(* CoDeSys 2.3.9.41 project: complex.pro *)
(* Libraries: ComService.lib 12.2.21 13:39:42, SysLibCom.lib 12.2.21 13:35:47, ModBus.lib 12.2.21 13:36:21, Util.lib 18.5.10 15:14:28, STANDARD.LIB 4.10.05 11:14:46, IECSFC.LIB 13.4.06 15:51:28, SYSLIBTIME.LIB 12.2.21 13:34:31, SYSTASKINFO.LIB 20.2.06 13:31:38, ANALYZATION.LIB 5.10.99 09:05:06, SYSLIBCALLBACK.LIB 20.2.06 13:31:08 *)

(* PLC configuration (modules and I/O channels)
Discrete input 8 bit [ID100] node 0, in %IB0 out %QB0 {Filtrationtime = 10; Filtrationtime = 10; Filtrationtime = 10; Filtrationtime = 10; Filtrationtime = 10; Filtrationtime = 10; Filtrationtime = 10; Filtrationtime = 10; Visibility = No; PinCount = 8; WatchDogPeriod = 1000; PollPeriod = 1}
  AT %IB0.0 [ByteInput] 8 discrete inputs
Discrete output - relay [ID102] node 1, in %IB1 out %QB1 {PinCount = 1; SafeValueBool = FALSE; Visibility = No}
  AT %QX1.0 [BitOutput] relay
Discrete output - relay [ID102] node 2, in %IB2 out %QB2 {PinCount = 1; SafeValueBool = FALSE; Visibility = No}
  AT %QX2.0 [BitOutput] relay
Discrete output - relay [ID102] node 3, in %IB3 out %QB3 {PinCount = 1; SafeValueBool = FALSE; Visibility = No}
  AT %QX3.0 [BitOutput] relay
Discrete output - relay [ID102] node 4, in %IB4 out %QB4 {PinCount = 1; SafeValueBool = FALSE; Visibility = No}
  AT %QX4.0 [BitOutput] relay
Discrete output - relay [ID102] node 5, in %IB5 out %QB5 {PinCount = 1; SafeValueBool = FALSE; Visibility = No}
  AT %QX5.0 [BitOutput] relay
Discrete output - relay [ID102] node 6, in %IB6 out %QB6 {PinCount = 1; SafeValueBool = FALSE; Visibility = No}
  AT %QX6.0 [BitOutput] relay
AT %QX7.0 [BitOutput] Special output
*)

(* Global variable list: Global_Variables *)
VAR_GLOBAL
	port_opened:  BYTE := 0;
	Settings:COMSETTINGS;
      	com_num: PORTS:=0;
	COM_SERVICE1: COM_SERVICE;

	port_opened2:  BYTE := 0;
	Settings2:COMSETTINGS;
      	com_num2: PORTS:=1;
	COM_SERVICE2: COM_SERVICE;


	ModBusWriteMultiReg232: MB_WR_REGS;
      ModBusReadHoldReg232: ARRAY[0..10] OF MB_RD_HOLD_REGS;
	TonConnect232:ARRAY[0..10] OF  TON;
	ToffConnect232:ARRAY[0..10] OF  TOF;
	ConnectionStatus232:ARRAY[0..10] OF  BOOL;
	Buffer232: ARRAY[0..255] OF BYTE;
	Cmpl232: ARRAY[0..10] OF BOOL;
	Err232: ARRAY[0..10] OF BYTE;
       SCADAData:ARRAY[0..70] OF WORD;

	Buffer: ARRAY[0..255] OF BYTE;

	Cmpl: ARRAY[0..30] OF BOOL;

	Err: ARRAY[0..30] OF BYTE;

	i: BYTE;
	j: BYTE;

      TonConnect: ARRAY[0..5] OF TON;
	ToffConnect: ARRAY[0..5] OF TOF;
	ConnectionStatus: ARRAY [0..5] OF BOOL;
      TimeOut: TIME := T#10ms;
(*****************************************************)
	KM1_2SET: INT;
	KM3_4SET: INT;
	KM5_6SET: INT;
	KM7SET: INT;
	KM8SET: INT;
	KM9SET: INT;
	KM10_11SET: INT;
	KM12_13SET: INT;
	KM14_16SET: INT;
	KM16SET: INT;
	KM17SET: INT;
	KM18SET: INT;
	KM19_20SET: INT;
	KM21_22SET: INT;
	KM23_24SET: INT;
	KM25_26SET: INT;
	KM27_28SET: INT;
	KM29SET: INT;
       KM30SET: INT;

(*****************************************************)
       DelayKM1_2: TIME;
	DelayKM3_4: TIME;
	DelayKM5_6: TIME;
	DelayKM7: TIME;
	DelayKM8: TIME;
	DelayKM9: TIME;
	DelayKM10_11: TIME;
	DelayKM12_13: TIME;
	DelayKM14_15: TIME;
	DelayKM16: TIME;
	DelayKM17: TIME;
	DelayKM18: TIME;
	DelayKM19_20: TIME;
	DelayKM21_22: TIME;
	DelayKM23_24: TIME;
	DelayKM25_26: TIME;
	DelayKM27_28: TIME;
	DelayKM29: TIME;
	DelayKM30: TIME;
(*****************************************************)


	ModBusWriteMultiCoil: ARRAY[0..1] OF MB_WR_COILS;
	ModBusReadHoldReg: ARRAY[0..10] OF MB_RD_HOLD_REGS;
	ModBusWriteMultiReg: ARRAY[0..10] OF MB_WR_REGS;
      NumberSend: BYTE;
      NumberSend2: BYTE;
	DisplayData:ARRAY[0..100] OF WORD;
       In1: WORD;
	In2: WORD;
	In3: WORD;
	In4: WORD;
	In5: WORD;

	Out1: WORD;
	Out2: WORD;
	Out3: WORD;
	Out4: WORD;
	Out5: WORD;


END_VAR

(* POU PLC_PRG, ST *)
PROGRAM PLC_PRG
VAR
       razrTON1: TON;
       nasTON: TON;
	errTON1: TON;
      errTON2: TON;
	trig: R_TRIG;

	start: BOOL;
	flash:BOOL;
END_VAR
IF start=0 THEN
Init();						(*	Открытие порта RS-485	*)
Init232();
start:=1;
END_IF
DelaySettings();
debug();
DenyList();
Link();
(* разр. работы*)
IF In2.0=FALSE OR In2.1=FALSE OR In2.2=FALSE OR In2.3=FALSE OR In2.4=FALSE
OR In2.5=FALSE OR In2.6=FALSE OR In2.7=FALSE OR In2.8=FALSE OR In2.9=FALSE OR In2.10=FALSE OR In2.11=FALSE
OR In2.12=FALSE OR In2.13=FALSE OR In2.14=FALSE OR In2.15=FALSE
OR In3.3=FALSE OR In3.4=FALSE OR In3.5=FALSE
OR Err[0]>0 OR Err[1]>0 OR Err[2]>0 OR Err[3]>0 OR Err[4]>0
(*OR (In5.4=TRUE AND In3.1=FALSE) *)THEN
Out4.5:=TRUE;
ELSE
Out4.5:=FALSE;
END_IF
IF In5.6 THEN
DisplayData[11].4:=FALSE;
DisplayData[63].7:=TRUE;
Out4.6:=TRUE;
(*trigLIGHT(CLK:=In5.6);
IF trigLIGHT.Q THEN
Out4.5:=FALSE;
END_IF*)
(*IF In2.0=FALSE OR In2.1=FALSE OR In2.2=FALSE OR In2.3=FALSE OR In2.4=FALSE
OR In2.5=FALSE OR In2.6=FALSE OR In2.7=FALSE OR In2.8=FALSE OR In2.9=FALSE OR In2.10=FALSE OR In2.11=FALSE
OR In2.12=FALSE OR In2.13=FALSE OR In2.14=FALSE OR In2.15=FALSE
OR In3.3=FALSE OR In3.4=FALSE OR In3.5=FALSE
OR Err[0]>0 OR Err[1]>0 OR Err[2]>0 OR Err[3]>0 OR Err[4]>0
(*OR (In5.4=TRUE AND In3.1=FALSE) *)THEN
Out4.5:=TRUE;
ELSE
Out4.5:=FALSE;
END_IF *)

ELSE
DisplayData[11].4:=TRUE;
DisplayData[63].7:=FALSE;
Out1:=0;
Out2.0:=FALSE;
Out2.1:=FALSE;
Out2.10:=FALSE;
Out2.11:=FALSE;
razrTON1(IN:=In5.6=FALSE, PT:=T#700ms);
IF razrTON1.Q=TRUE THEN
IF Out4.6=FALSE THEN
Out4.6:=TRUE;
razrTON1(In:=FALSE);
ELSE
Out4.6:=FALSE;
razrTON1(In:=FALSE);
END_IF
END_IF
(*IF In2.0=FALSE OR In2.1=FALSE OR In2.2=FALSE OR In2.3=FALSE OR In2.4=FALSE
OR In2.5=FALSE OR In2.6=FALSE OR In2.7=FALSE OR In2.8=FALSE OR In2.9=FALSE OR In2.10=FALSE OR In2.11=FALSE
OR In2.12=FALSE OR In2.13=FALSE OR In2.14=FALSE OR In2.15=FALSE
OR In3.3=FALSE OR In3.4=FALSE OR In3.5=FALSE OR Err[0]>0 OR Err[1]>0 OR Err[2]>0 OR Err[3]>0 OR Err[4]>0 THEN
(*razrTON1(IN:=In5.6=FALSE, PT:=T#500ms);*)
Out4.6:=TRUE;
ELSE
IF razrTON1.Q=TRUE THEN
IF Out4.6=FALSE THEN
Out4.6:=TRUE;
razrTON1(In:=FALSE);
ELSE
Out4.6:=FALSE;
razrTON1(In:=FALSE);
END_IF
END_IF
END_IF*)

END_IF

(*ОТОБР. РЕЖИМОВ *)
IF In5.9 THEN (*Люди*)
DisplayData[11].2:=TRUE;
ELSE
DisplayData[11].2:=FALSE;
END_IF
IF In5.10 THEN (*Груз*)
DisplayData[11].3:=TRUE;
ELSE
DisplayData[11].3:=FALSE;
END_IF
IF In5.11 THEN (*Негабарит*)
DisplayData[11].0:=TRUE;
ELSE
DisplayData[11].0:=FALSE;
END_IF
IF In5.9=FALSE AND In5.10=FALSE AND In5.11=FALSE THEN (* Ревизия *)
DisplayData[11].1:=TRUE;
ELSE
DisplayData[11].1:=FALSE;
END_IF
(* противопож двери*)
IF In2.12=TRUE AND In5.2=TRUE THEN (*ДВЕРИ 1 *)
Out2.2:=TRUE;
ELSE
Out2.2:=FALSE;
(*DisplayData[16].3:=FALSE;*)
END_IF
IF In2.12=TRUE AND In5.3=TRUE THEN
Out2.3:=TRUE;
ELSE
Out2.3:=FALSE;
(*DisplayData[16].3:=FALSE;*)
END_IF

IF In2.13=TRUE AND In3.6=TRUE THEN (*ДВЕРИ 2 *)
Out2.4:=TRUE;
ELSE
Out2.4:=FALSE;
(*DisplayData[16].4:=FALSE; *)
END_IF
IF In2.13=TRUE AND In3.7=TRUE THEN
Out2.5:=TRUE;
ELSE
Out2.5:=FALSE;
(*DisplayData[16].4:=FALSE; *)
END_IF


IF In2.14=TRUE AND In3.8=TRUE THEN (*ДВЕРИ 3 *)
Out2.6:=TRUE;
ELSE
Out2.6:=FALSE;
(*DisplayData[16].5:=FALSE; *)
END_IF
IF In2.13=TRUE AND In3.9=TRUE THEN
Out2.7:=TRUE;
ELSE
Out2.7:=FALSE;
(*DisplayData[16].5:=FALSE;*)
END_IF

IF In2.14=TRUE AND In3.10=TRUE THEN (*ДВЕРИ 4 *)
Out2.8:=TRUE;
ELSE
Out2.8:=FALSE;
(*DisplayData[16].6:=FALSE;*)
END_IF
IF In2.13=TRUE AND In3.11=TRUE THEN
Out2.9:=TRUE;
ELSE
Out2.9:=FALSE;
(*DisplayData[16].6:=FALSE;*)
END_IF



IF In5.4 AND In5.6 AND In3.4 THEN (* НАСОС *)
errTON2(IN:=In5.4, PT:=t#500ms);
IF errTON2.Q=FALSE AND In3.1=FALSE THEN
Out2.12:=TRUE;
ELSIF errTON2.Q=TRUE AND In3.1=FALSE THEN
Out2.12:=FALSE;
Out4.4:=FALSE;
Out4.5:=TRUE;
ELSIF errTON2.Q=TRUE AND In3.1=TRUE THEN
Out2.12:=TRUE;
Out4.4:=TRUE;
END_IF

END_IF

IF In3.1 THEN
Out4.4:=TRUE;
END_IF

IF In5.5=FALSE OR In5.6=FALSE OR In3.4=FALSE THEN
errTON2(IN:=FALSE);
trig(CLK:=In5.6=FALSE);
Out2.12:=FALSE;
Out4.4:=FALSE;
IF trig.Q THEN
Out4.5:=FALSE;
END_IF
END_IF
(*********************************************************************************************************)
(* РЕЖИМ ЛЮДИ *)
IF In5.9 AND In5.6 THEN
(*DisplayData[11].2:=TRUE;*)

IF in4.8 THEN (*кулаки лев*)
Out1.8:=TRUE;
ELSE
Out1.8:=FALSE;
END_IF
IF In4.2 AND In5.14 THEN (*двери лев*)
Out1.2:=TRUE;
ELSE
Out1.2:=FALSE;
END_IF
IF In4.3 AND In5.14 THEN
Out1.3:=TRUE;
ELSE
Out1.3:=FALSE;
END_IF
IF in5.1 THEN (*кулаки прав*)
Out2.1:=TRUE;
ELSE
Out2.1:=FALSE;
END_IF
IF In4.11 AND In5.15 THEN (*двери прав*)
Out1.11:=TRUE;
ELSE
Out1.11:=FALSE;
END_IF
IF In4.12 AND In5.15 THEN
Out1.12:=TRUE;
ELSE
Out1.12:=FALSE;
END_IF

(*ELSE
DisplayData[11].2:=FALSE; *)
END_IF
(*********************************************************************************************************)
(* РЕЖИМ ГРУЗ *)
IF In5.10 AND In5.6 THEN

IF In3.12=TRUE AND In3.3=TRUE THEN (*ЛЕБЕДКА *)
Out2.10:=TRUE;
ELSE
Out2.10:=FALSE;
(*DisplayData[16].3:=FALSE;*)
END_IF
IF In3.13=TRUE AND In3.3=TRUE THEN
Out2.11:=TRUE;
ELSE
Out2.11:=FALSE;
(*DisplayData[16].3:=FALSE;*)
END_IF


(*DisplayData[11].3:=TRUE;*)
IF in4.8 THEN (*кулаки лев*)
Out1.8:=TRUE;
ELSE
Out1.8:=FALSE;
END_IF
IF In4.2 AND In5.14 THEN (*двери лев*)
Out1.2:=TRUE;
ELSE
Out1.2:=FALSE;
END_IF
IF In4.3 AND In5.14 THEN
Out1.3:=TRUE;
ELSE
Out1.3:=FALSE;
END_IF
IF In4.0 AND In5.14 THEN (*толкатель лев*)
Out1.0:=TRUE;
ELSE
Out1.0:=FALSE;
END_IF
IF In4.1 AND In5.14 THEN
Out1.1:=TRUE;
ELSE
Out1.1:=FALSE;
END_IF
IF In4.4 AND In5.14 THEN (*стопора предкл. лев*)
Out1.4:=TRUE;
ELSE
Out1.4:=FALSE;
END_IF
IF In4.5 AND In5.14 THEN
Out1.5:=TRUE;
ELSE
Out1.5:=FALSE;
END_IF
IF In4.6 AND In5.14 THEN (*стопора вход лев*)
Out1.6:=TRUE;
ELSE
Out1.6:=FALSE;
END_IF
IF In4.7 AND In5.14 THEN (*стопора доз лев*)
Out1.7:=TRUE;
ELSE
Out1.7:=FALSE;
END_IF
IF in5.1 THEN (*кулаки прав*)
Out2.1:=TRUE;
ELSE
Out2.1:=FALSE;
END_IF
IF In4.11 AND In5.15 THEN (*двери прав*)
Out1.11:=TRUE;
ELSE
Out1.11:=FALSE;
END_IF
IF In4.12 AND In5.15 THEN
Out1.12:=TRUE;
ELSE
Out1.12:=FALSE;
END_IF
IF In4.9 AND In5.15 THEN (*толкатель прав*)
Out1.9:=TRUE;
ELSE
Out1.9:=FALSE;
END_IF
IF In4.10 AND In5.15 THEN
Out1.10:=TRUE;
ELSE
Out1.10:=FALSE;
END_IF
IF In4.13 AND In5.15 THEN (*стопора предкл. прав*)
Out1.13:=TRUE;
ELSE
Out1.13:=FALSE;
END_IF
IF In4.14 AND In5.15 THEN
Out1.14:=TRUE;
ELSE
Out1.14:=FALSE;
END_IF
IF In4.15 AND In5.15 THEN (*стопора вход прав*)
Out1.15:=TRUE;
ELSE
Out1.15:=FALSE;
END_IF
IF In5.0 AND In5.15 THEN (*стопора доз прав*)
Out2.0:=TRUE;
ELSE
Out2.0:=FALSE;
END_IF

(*ELSE
DisplayData[11].3:=FALSE; *)

END_IF
(*********************************************************************************************************)
(* РЕЖИМ НЕГАБАРИТ *)
IF In5.11  AND In5.6 THEN
(*DisplayData[11].0:=TRUE;*)

IF In3.12=TRUE AND In3.3=TRUE THEN (*ЛЕБЕДКА *)
Out2.10:=TRUE;
ELSE
Out2.10:=FALSE;
(*DisplayData[16].3:=FALSE;*)
END_IF
IF In3.13=TRUE AND In3.3=TRUE THEN
Out2.11:=TRUE;
ELSE
Out2.11:=FALSE;
(*DisplayData[16].3:=FALSE;*)
END_IF

IF in4.8 THEN (*кулаки лев*)
Out1.8:=TRUE;
ELSE
Out1.8:=FALSE;
END_IF
IF In4.2 THEN (*двери лев*)
Out1.2:=TRUE;
ELSE
Out1.2:=FALSE;
END_IF
IF In4.3 THEN
Out1.3:=TRUE;
ELSE
Out1.3:=FALSE;
END_IF
IF In4.0 AND In5.14 THEN (*толкатель лев*)
Out1.0:=TRUE;
ELSE
Out1.0:=FALSE;
END_IF
IF In4.1 AND In5.14 THEN
Out1.1:=TRUE;
ELSE
Out1.1:=FALSE;
END_IF
IF In4.4 AND In5.14 THEN (*стопора предкл. лев*)
Out1.4:=TRUE;
ELSE
Out1.4:=FALSE;
END_IF
IF In4.5 AND In5.14 THEN
Out1.5:=TRUE;
ELSE
Out1.5:=FALSE;
END_IF
IF In4.6 AND In5.14 THEN (*стопора вход лев*)
Out1.6:=TRUE;
ELSE
Out1.6:=FALSE;
END_IF
IF In4.7 AND In5.14 THEN (*стопора доз лев*)
Out1.7:=TRUE;
ELSE
Out1.7:=FALSE;
END_IF
IF in5.1 THEN (*кулаки прав*)
Out2.1:=TRUE;
ELSE
Out2.1:=FALSE;
END_IF
IF In4.11 THEN (*двери прав*)
Out1.11:=TRUE;
ELSE
Out1.11:=FALSE;
END_IF
IF In4.12 THEN
Out1.12:=TRUE;
ELSE
Out1.12:=FALSE;
END_IF
IF In4.9 AND In5.15 THEN (*толкатель прав*)
Out1.9:=TRUE;
ELSE
Out1.9:=FALSE;
END_IF
IF In4.10 AND In5.15 THEN
Out1.10:=TRUE;
ELSE
Out1.10:=FALSE;
END_IF
IF In4.13 AND In5.15 THEN (*стопора предкл. прав*)
Out1.13:=TRUE;
ELSE
Out1.13:=FALSE;
END_IF
IF In4.14 AND In5.15 THEN
Out1.14:=TRUE;
ELSE
Out1.14:=FALSE;
END_IF
IF In4.15 AND In5.15 THEN (*стопора вход прав*)
Out1.15:=TRUE;
ELSE
Out1.15:=FALSE;
END_IF
IF In5.0 AND In5.15 THEN (*стопора доз прав*)
Out2.0:=TRUE;
ELSE
Out2.0:=FALSE;
END_IF

(*ELSE
DisplayData[11].0:=FALSE; *)
END_IF
(*********************************************************************************************************)
(* РЕЖИМ РЕВИЗИЯ *)
IF In5.9=FALSE AND In5.10=FALSE AND In5.11=FALSE AND In5.6 THEN
(*DisplayData[11].1:=TRUE;*)

IF in4.8 THEN (*кулаки лев*)
Out1.8:=TRUE;
ELSE
Out1.8:=FALSE;
END_IF
IF In4.2 AND In5.14 THEN (*двери лев*)
Out1.2:=TRUE;
ELSE
Out1.2:=FALSE;
END_IF
IF In4.3 AND In5.14 THEN
Out1.3:=TRUE;
ELSE
Out1.3:=FALSE;
END_IF
IF in5.1 THEN (*кулаки прав*)
Out2.1:=TRUE;
ELSE
Out2.1:=FALSE;
END_IF
IF In4.11 AND In5.15 THEN (*двери прав*)
Out1.11:=TRUE;
ELSE
Out1.11:=FALSE;
END_IF
IF In4.12 AND In5.15 THEN
Out1.12:=TRUE;
ELSE
Out1.12:=FALSE;
END_IF

(*ELSE
DisplayData[11].1:=FALSE;*)
END_IF
(*********************************************************************************************************)
IF  In5.12 AND In5.12 THEN (*КУЛАКИ ЛЕВ*)
DisplayData[11].5:=TRUE;
Out4.0:=TRUE;
ELSE
DisplayData[11].5:=FALSE;
Out4.0:=FALSE;
END_IF

IF  In5.13 AND In5.13 THEN (* КУЛАКИ ПРАВ *)
DisplayData[11].7:=TRUE;
Out4.2:=TRUE;
ELSE
DisplayData[11].7:=FALSE;
Out4.2:=FALSE;
END_IF

IF In5.14=TRUE AND In5.11=FALSE THEN  (* ПРИХОД КЛЕТИ ЛЕВ *)
DisplayData[11].6:=TRUE;
Out4.1:=TRUE;
ELSIF In5.14=FALSE AND In5.11=FALSE THEN
DisplayData[11].6:=FALSE;
Out4.1:=FALSE;
ELSIF In5.14=TRUE AND In5.11=TRUE THEN
DisplayData[11].6:=TRUE;
Out4.1:=TRUE;
ELSIF In5.14=FALSE AND In5.11=TRUE THEN
DisplayData[11].6:=FALSE;
Out4.1:=TRUE;
END_IF

IF In5.15 =TRUE AND In5.11=FALSE THEN  (* ПРИХОД КЛЕТИ ПРАВ *)
DisplayData[11].8:=TRUE;
Out4.3:=TRUE;
ELSIF In5.15=FALSE AND In5.11=FALSE THEN
DisplayData[11].8:=FALSE;
Out4.3:=FALSE;
ELSIF In5.15=TRUE AND In5.11=TRUE THEN
DisplayData[11].8:=TRUE;
Out4.3:=TRUE;
ELSIF In5.15=FALSE AND In5.11=TRUE THEN
DisplayData[11].8:=FALSE;
Out4.3:=TRUE;
END_IF
END_PROGRAM

(* POU Init, ST *)
FUNCTION Init : BOOL
VAR_INPUT
END_VAR
VAR
END_VAR
WHILE port_opened=0 DO
	IF port_opened=0 THEN
		Settings.Port:=com_num;
		Settings.dwBaudRate:=57600;
		Settings.byParity:=0;
		Settings.dwTimeout:=0;
		Settings.byStopBits:=0;
		Settings.dwBufferSize:=0;
		Settings.dwScan:=0;
	END_IF
	COM_SERVICE1(Enable:=(port_opened=0) , Settings:=Settings , Task:=OPEN_TSK  );
	IF COM_SERVICE1.ready THEN
		port_opened:=2;
	END_IF
END_WHILE
END_FUNCTION

(* POU Init232, ST *)
FUNCTION Init232 : BOOL
VAR_INPUT
END_VAR
VAR
	PultWork: BOOL;
END_VAR
PultWork;
(*WHILE port_opened2=0 DO
	IF port_opened2=0 THEN
		Settings2.Port:=com_num2;
		Settings2.dwBaudRate:=19200;
		Settings2.byParity:=0;
		Settings2.dwTimeout:=0;
		Settings2.byStopBits:=0;
		Settings2.dwBufferSize:=0;
		Settings2.dwScan:=0;
	END_IF
	COM_SERVICE2(Enable:=(port_opened2=0) , Settings:=Settings2 , Task:=OPEN_TSK  );
	IF COM_SERVICE2.ready THEN
		port_opened2:=2;
	END_IF
END_WHILE*)
END_FUNCTION

(* POU DelaySettings, ST *)
FUNCTION DelaySettings : BOOL
VAR_INPUT
END_VAR
VAR
END_VAR
(* delay settings *)




DelayKM1_2;
END_FUNCTION

(* POU debug, ST *)
FUNCTION debug : BOOL
VAR_INPUT
END_VAR
VAR
END_VAR
(************- INPUTS -***************)
DisplayData[0].0:=In1.0;
DisplayData[0].1:=In1.1;
DisplayData[0].2:=In1.2;
DisplayData[0].3:=In1.3;
DisplayData[0].4:=In1.4;
DisplayData[0].5:=In1.5;
DisplayData[0].6:=In1.6;
DisplayData[0].7:=In1.7;
DisplayData[0].8:=In1.8;
DisplayData[0].9:=In1.9;
DisplayData[0].10:=In1.10;
DisplayData[0].11:=In1.11;
DisplayData[0].12:=In1.12;
DisplayData[0].13:=In1.13;
DisplayData[0].14:=In1.14;
DisplayData[0].15:=In1.15;
(***************************)
DisplayData[2].0:=In2.0;
DisplayData[2].1:=In2.1;
DisplayData[2].2:=In2.2;
DisplayData[2].3:=In2.3;
DisplayData[2].4:=In2.4;
DisplayData[2].5:=In2.5;
DisplayData[2].6:=In2.6;
DisplayData[2].7:=In2.7;
DisplayData[2].8:=In2.8;
DisplayData[2].9:=In2.9;
DisplayData[2].10:=In2.10;
DisplayData[2].11:=In2.11;
DisplayData[2].12:=In2.12;
DisplayData[2].13:=In2.13;
DisplayData[2].14:=In2.14;
DisplayData[2].15:=In2.15;
(***************************)
DisplayData[4].0:=In3.0;
DisplayData[4].1:=In3.1;
DisplayData[4].2:=In3.2;
DisplayData[4].3:=In3.3;
DisplayData[4].4:=In3.4;
DisplayData[4].5:=In3.5;
DisplayData[4].6:=In3.6;
DisplayData[4].7:=In3.7;
DisplayData[4].8:=In3.8;
DisplayData[4].9:=In3.9;
DisplayData[4].10:=In3.10;
DisplayData[4].11:=In3.11;
DisplayData[4].12:=In3.12;
DisplayData[4].13:=In3.13;
DisplayData[4].14:=In3.14;
DisplayData[4].15:=In3.15;
(***************************)
DisplayData[6].0:=In4.0;
DisplayData[6].1:=In4.1;
DisplayData[6].2:=In4.2;
DisplayData[6].3:=In4.3;
DisplayData[6].4:=In4.4;
DisplayData[6].5:=In4.5;
DisplayData[6].6:=In4.6;
DisplayData[6].7:=In4.7;
DisplayData[6].8:=In4.8;
DisplayData[6].9:=In4.9;
DisplayData[6].10:=In4.10;
DisplayData[6].11:=In4.11;
DisplayData[6].12:=In4.12;
DisplayData[6].13:=In4.13;
DisplayData[6].14:=In4.14;
DisplayData[6].15:=In4.15;
(***************************)
DisplayData[8].0:=In5.0;
DisplayData[8].1:=In5.1;
DisplayData[8].2:=In5.2;
DisplayData[8].3:=In5.3;
DisplayData[8].4:=In5.4;
DisplayData[8].5:=In5.5;
DisplayData[8].6:=In5.6;
DisplayData[8].7:=In5.7;
DisplayData[8].8:=In5.8;
DisplayData[8].9:=In5.9;
DisplayData[8].10:=In5.10;
DisplayData[8].11:=In5.11;
DisplayData[8].12:=In5.12;
DisplayData[8].13:=In5.13;
DisplayData[8].14:=In5.14;
DisplayData[8].15:=In5.15;
(********************************************************************************************************)
(**************-OUTPUTS -*************)
DisplayData[1].0:=Out1.0;
DisplayData[1].1:=Out1.1;
DisplayData[1].2:=Out1.2;
DisplayData[1].3:=Out1.3;
DisplayData[1].4:=Out1.4;
DisplayData[1].5:=Out1.5;
DisplayData[1].6:=Out1.6;
DisplayData[1].7:=Out1.7;
DisplayData[1].8:=Out1.8;
DisplayData[1].9:=Out1.9;
DisplayData[1].10:=Out1.10;
DisplayData[1].11:=Out1.11;
DisplayData[1].12:=Out1.12;
DisplayData[1].13:=Out1.13;
DisplayData[1].14:=Out1.14;
DisplayData[1].15:=Out1.15;
(***************************)
DisplayData[3].0:=Out2.0;
DisplayData[3].1:=Out2.1;
DisplayData[3].2:=Out2.2;
DisplayData[3].3:=Out2.3;
DisplayData[3].4:=Out2.4;
DisplayData[3].5:=Out2.5;
DisplayData[3].6:=Out2.6;
DisplayData[3].7:=Out2.7;
DisplayData[3].8:=Out2.8;
DisplayData[3].9:=Out2.9;
DisplayData[3].10:=Out2.10;
DisplayData[3].11:=Out2.11;
DisplayData[3].12:=Out2.12;
DisplayData[3].13:=Out2.13;
DisplayData[3].14:=Out2.14;
DisplayData[3].15:=Out2.15;
(***************************)
DisplayData[5].0:=Out3.0;
DisplayData[5].1:=Out3.1;
DisplayData[5].2:=Out3.2;
DisplayData[5].3:=Out3.3;
DisplayData[5].4:=Out3.4;
DisplayData[5].5:=Out3.5;
DisplayData[5].6:=Out3.6;
DisplayData[5].7:=Out3.7;
DisplayData[5].8:=Out3.8;
DisplayData[5].9:=Out3.9;
DisplayData[5].10:=Out3.10;
DisplayData[5].11:=Out3.11;
DisplayData[5].12:=Out3.12;
DisplayData[5].13:=Out3.13;
DisplayData[5].14:=Out3.14;
DisplayData[5].15:=Out3.15;
(***************************)
DisplayData[7].0:=Out4.0;
DisplayData[7].1:=Out4.1;
DisplayData[7].2:=Out4.2;
DisplayData[7].3:=Out4.3;
DisplayData[7].4:=Out4.4;
DisplayData[7].5:=Out4.5;
DisplayData[7].6:=Out4.6;
DisplayData[7].7:=Out4.7;
DisplayData[7].8:=Out4.8;
DisplayData[7].9:=Out4.9;
DisplayData[7].10:=Out4.10;
DisplayData[7].11:=Out4.11;
DisplayData[7].12:=Out4.12;
DisplayData[7].13:=Out4.13;
DisplayData[7].14:=Out4.14;
DisplayData[7].15:=Out4.15;
(***************************)
DisplayData[9].0:=Out5.0;
DisplayData[9].1:=Out5.1;
DisplayData[9].2:=Out5.2;
DisplayData[9].3:=Out5.3;
DisplayData[9].4:=Out5.4;
DisplayData[9].5:=Out5.5;
DisplayData[9].6:=Out5.6;
DisplayData[9].7:=Out5.7;
DisplayData[9].8:=Out5.8;
DisplayData[9].9:=Out5.9;
DisplayData[9].10:=Out5.10;
DisplayData[9].11:=Out5.11;
DisplayData[9].12:=Out5.12;
DisplayData[9].13:=Out5.13;
DisplayData[9].14:=Out5.14;
DisplayData[9].15:=Out5.15;
(***********МТЗ ЛЕВ КЛЕТЬ*************)
IF In2.0 THEN
DisplayData[12].9:=FALSE;
ELSE
DisplayData[12].9:=TRUE;
DisplayData[15].0:=FALSE;
Out1.0:=FALSE;
Out1.1:=FALSE;
END_IF
IF In2.1 THEN
DisplayData[12].10:=FALSE;
ELSE
DisplayData[12].10:=TRUE;
DisplayData[15].1:=FALSE;
Out1.2:=FALSE;
Out1.3:=FALSE;
END_IF
IF In2.2 THEN
DisplayData[12].11:=FALSE;
ELSE
DisplayData[12].11:=TRUE;
DisplayData[15].2:=FALSE;
Out1.4:=FALSE;
Out1.5:=FALSE;
END_IF
IF In2.3 THEN
DisplayData[12].12:=FALSE;
ELSE
DisplayData[12].12:=TRUE;
DisplayData[15].3:=FALSE;
Out1.6:=FALSE;
END_IF
IF In2.4 THEN
DisplayData[12].13:=FALSE;
ELSE
DisplayData[12].13:=TRUE;
DisplayData[15].4:=FALSE;
Out1.7:=FALSE;
END_IF
IF In2.5 THEN
DisplayData[12].14:=FALSE;
ELSE
DisplayData[12].14:=TRUE;
DisplayData[15].5:=FALSE;
Out1.8:=FALSE;
END_IF
(***********МТЗ ПРАВ КЛЕТЬ*************)
IF In2.6 THEN
DisplayData[13].9:=FALSE;
ELSE
DisplayData[13].9:=TRUE;
DisplayData[15].6:=FALSE;
Out1.9:=FALSE;
Out1.10:=FALSE;
END_IF
IF In2.7 THEN
DisplayData[13].10:=FALSE;
ELSE
DisplayData[13].10:=TRUE;
DisplayData[15].7:=FALSE;
Out1.11:=FALSE;
Out1.12:=FALSE;
END_IF
IF In2.8 THEN
DisplayData[13].11:=FALSE;
ELSE
DisplayData[13].11:=TRUE;
DisplayData[15].8:=FALSE;
Out1.13:=FALSE;
Out1.14:=FALSE;
END_IF
IF In2.9 THEN
DisplayData[13].12:=FALSE;
ELSE
DisplayData[13].12:=TRUE;
DisplayData[15].9:=FALSE;
Out1.15:=FALSE;
END_IF
IF In2.10 THEN
DisplayData[13].13:=FALSE;
ELSE
DisplayData[13].13:=TRUE;
DisplayData[15].10:=FALSE;
Out2.0:=FALSE;
END_IF
IF In2.11 THEN
DisplayData[13].14:=FALSE;
ELSE
DisplayData[13].14:=TRUE;
DisplayData[15].11:=FALSE;
Out2.1:=FALSE;
END_IF
(***********МТЗ ВСП МЕХАНИЗМЫ*************)
IF In3.3 THEN
DisplayData[16].7:=FALSE;
ELSE
DisplayData[16].7:=TRUE;
DisplayData[16].0:=FALSE;
Out2.10:=FALSE;
Out2.11:=FALSE;
END_IF
IF In3.4 THEN
DisplayData[16].8:=FALSE;
ELSE
DisplayData[16].8:=TRUE;
DisplayData[16].1:=FALSE;
Out2.12:=FALSE;
END_IF
IF In3.5 THEN
DisplayData[16].9:=FALSE;
ELSE
DisplayData[16].9:=TRUE;
DisplayData[16].2:=FALSE;
Out2.13:=FALSE;
END_IF
IF In2.12 THEN
DisplayData[16].10:=FALSE;
ELSE
DisplayData[16].10:=TRUE;
DisplayData[16].3:=FALSE;
Out2.2:=FALSE;
Out2.3:=FALSE;
END_IF
IF In2.13 THEN
DisplayData[16].11:=FALSE;
ELSE
DisplayData[16].11:=TRUE;
DisplayData[16].4:=FALSE;
Out2.4:=FALSE;
Out2.5:=FALSE;
END_IF
IF In2.14 THEN
DisplayData[16].12:=FALSE;
ELSE
DisplayData[16].12:=TRUE;
DisplayData[16].5:=FALSE;
Out2.6:=FALSE;
Out2.7:=FALSE;
END_IF
IF In2.15 THEN
DisplayData[16].13:=FALSE;
ELSE
DisplayData[16].13:=TRUE;
DisplayData[16].6:=FALSE;
Out2.8:=FALSE;
Out2.9:=FALSE;
END_IF

(***********ПУСКИ  И ПОДТВ КМ ЛЕВ*************)
IF In2.0=TRUE THEN
IF In1.0 AND In4.0 THEN
DisplayData[12].0:=TRUE;
ELSE
DisplayData[12].0:=FALSE;
END_IF
IF In1.0 AND In4.1 THEN
DisplayData[12].1:=TRUE;
ELSE
DisplayData[12].1:=FALSE;
END_IF
DisplayData[15].0:=In4.0 OR In4.1 ;
END_IF

IF In2.1=TRUE THEN
IF In1.1 AND In4.2 THEN
DisplayData[12].15:=TRUE;
ELSE
DisplayData[12].15:=FALSE;
END_IF
IF In1.1 AND In4.3 THEN
DisplayData[12].3:=TRUE;
ELSE
DisplayData[12].3:=FALSE;
END_IF
DisplayData[15].1:=In4.2 OR In4.3;
END_IF

IF In2.2=TRUE THEN
IF In1.2 AND In4.4 THEN
DisplayData[12].4:=TRUE;
ELSE
DisplayData[12].4:=FALSE;
END_IF
IF In1.2 AND In4.5 THEN
DisplayData[12].5:=TRUE;
ELSE
DisplayData[12].5:=FALSE;
END_IF
DisplayData[15].2:=In4.4 OR In4.5;
END_IF

IF In2.3=TRUE THEN
DisplayData[12].6:=In1.3;
DisplayData[15].3:=In4.6;
END_IF

IF In2.4=TRUE THEN
DisplayData[12].7:=In1.4;
DisplayData[15].4:=In4.7;
END_IF

IF In2.5=TRUE THEN
DisplayData[12].8:=In1.5;
DisplayData[15].5:=In4.8;
END_IF

(***********ПУСКИ И ПОДТВ КМ ПРАВ*************)
IF In2.6=TRUE THEN
IF In1.6 AND In4.9 THEN
DisplayData[13].0:=TRUE;
ELSE
DisplayData[13].0:=FALSE;
END_IF
IF In1.6 AND In4.10 THEN
DisplayData[13].1:=TRUE;
ELSE
DisplayData[13].1:=FALSE;
END_IF
DisplayData[15].6:=In4.9 OR In4.10;
END_IF

IF In2.7=TRUE THEN
IF In1.7 AND In4.11 THEN
DisplayData[13].2:=TRUE;
ELSE
DisplayData[13].2:=FALSE;
END_IF
IF In1.7 AND In4.12 THEN
DisplayData[13].3:=TRUE;
ELSE
DisplayData[13].3:=FALSE;
END_IF
DisplayData[15].7:=In4.11 OR In4.12;
END_IF

IF In2.8=TRUE THEN
IF In1.8 AND In4.13 THEN
DisplayData[13].4:=TRUE;
ELSE
DisplayData[13].4:=FALSE;
END_IF
IF In1.8 AND In4.14 THEN
DisplayData[13].5:=TRUE;
ELSE
DisplayData[13].5:=FALSE;
END_IF
DisplayData[15].8:=In4.13 OR In4.14;
END_IF

IF In2.9=TRUE THEN
DisplayData[13].6:=In1.9;
DisplayData[15].9:=In4.15;
END_IF

IF In2.10=TRUE THEN
DisplayData[13].7:=In1.10;
DisplayData[15].10:=In5.0;
END_IF

IF In2.11=TRUE THEN
DisplayData[13].8:=In1.11;
DisplayData[15].11:=In5.1;
END_IF
(***********ПУСКИ И ПОДТВ КМ ВСП МЕХ*************)
IF In3.3=TRUE THEN
IF In3.0 AND In3.12 THEN
DisplayData[14].0:=TRUE;
ELSE
DisplayData[14].0:=FALSE;
END_IF
IF In3.0 AND In3.13 THEN
DisplayData[14].1:=TRUE;
ELSE
DisplayData[14].1:=FALSE;
END_IF
DisplayData[16].0:=In3.12 OR In3.13;

END_IF
(*IF In3.4=TRUE THEN
DisplayData[14].2:=In3.1;
DisplayData[16].1:=In5.4;
END_IF*)
DisplayData[14].2:=In3.1;
DisplayData[16].1:=In5.4;
(*IF In3.5=TRUE THEN                 РЕЗЕРВ
DisplayData[14].3:=
DisplayData[16].2:=In3.2; 
END_IF*)
IF In2.12=TRUE THEN
IF In1.12 AND In5.2 THEN
DisplayData[14].4:=TRUE;
ELSE
DisplayData[14].4:=FALSE;
END_IF
IF In1.12 AND In5.3 THEN
DisplayData[14].5:=TRUE;
ELSE
DisplayData[14].5:=FALSE;
END_IF
DisplayData[16].3:=In5.2 OR In5.3;
END_IF

IF In2.13=TRUE THEN
IF In1.13 AND In3.6 THEN
DisplayData[14].6:=TRUE;
ELSE
DisplayData[14].6:=FALSE;
END_IF
IF In1.13 AND In3.7 THEN
DisplayData[14].7:=TRUE;
ELSE
DisplayData[14].7:=FALSE;
END_IF
DisplayData[16].4:=In3.6 OR In3.7;
END_IF


IF In2.14=TRUE THEN
IF In1.14 AND In3.8 THEN
DisplayData[14].8:=TRUE;
ELSE
DisplayData[14].8:=FALSE;
END_IF
IF In1.14 AND In3.8 THEN
DisplayData[14].9:=TRUE;
ELSE
DisplayData[14].9:=FALSE;
END_IF
DisplayData[16].5:=In3.8 OR In3.9;
END_IF


IF In2.15=TRUE THEN
IF In1.15 AND In3.10 THEN
DisplayData[14].10:=TRUE;
ELSE
DisplayData[14].10:=FALSE;
END_IF
IF In1.15 AND In3.11 THEN
DisplayData[14].11:=TRUE;
ELSE
DisplayData[14].11:=FALSE;
END_IF
DisplayData[16].6:=In3.10 OR In3.11;
END_IF
END_FUNCTION

(* POU DenyList, ST *)
FUNCTION DenyList : BOOL
VAR_INPUT
END_VAR
VAR

END_VAR
(* МТЗ*)
IF In2.0=FALSE OR In2.1=FALSE OR In2.2=FALSE OR In2.3=FALSE OR In2.4=FALSE
OR In2.5=FALSE OR In2.6=FALSE OR In2.7=FALSE OR In2.8=FALSE OR In2.9=FALSE OR In2.10=FALSE OR In2.11=FALSE
OR In2.12=FALSE OR In2.13=FALSE OR In2.14=FALSE OR In2.15=FALSE
OR In3.3=FALSE OR In3.4=FALSE OR In3.5=FALSE THEN
DisplayData[60].0:=TRUE;
DisplayData[63].0:=FALSE;
ELSE
DisplayData[60].0:=FALSE;
DisplayData[63].0:=TRUE;
END_IF

IF In2.0=FALSE THEN
DisplayData[61].0:=TRUE;
ELSE
DisplayData[61].0:=FALSE;
END_IF
IF In2.1=FALSE THEN
DisplayData[61].1:=TRUE;
ELSE
DisplayData[61].1:=FALSE;
END_IF
IF In2.2=FALSE THEN
DisplayData[61].2:=TRUE;
ELSE
DisplayData[61].2:=FALSE;
END_IF
IF In2.3=FALSE THEN
DisplayData[61].3:=TRUE;
ELSE
DisplayData[61].3:=FALSE;
END_IF
IF In2.4=FALSE THEN
DisplayData[61].4:=TRUE;
ELSE
DisplayData[61].4:=FALSE;
END_IF
IF In2.5=FALSE THEN
DisplayData[61].5:=TRUE;
ELSE
DisplayData[61].5:=FALSE;
END_IF
IF In2.6=FALSE THEN
DisplayData[61].6:=TRUE;
ELSE
DisplayData[61].6:=FALSE;
END_IF
IF In2.7=FALSE THEN
DisplayData[61].7:=TRUE;
ELSE
DisplayData[61].7:=FALSE;
END_IF
IF In2.8=FALSE THEN
DisplayData[61].8:=TRUE;
ELSE
DisplayData[61].8:=FALSE;
END_IF
IF In2.9=FALSE THEN
DisplayData[61].9:=TRUE;
ELSE
DisplayData[61].9:=FALSE;
END_IF
IF In2.10=FALSE THEN
DisplayData[61].10:=TRUE;
ELSE
DisplayData[61].10:=FALSE;
END_IF
IF In2.11=FALSE THEN
DisplayData[61].11:=TRUE;
ELSE
DisplayData[61].11:=FALSE;
END_IF
IF In2.12=FALSE THEN
DisplayData[61].12:=TRUE;
ELSE
DisplayData[61].12:=FALSE;
END_IF
IF In2.13=FALSE THEN
DisplayData[61].13:=TRUE;
ELSE
DisplayData[61].13:=FALSE;
END_IF
IF In2.14=FALSE THEN
DisplayData[61].14:=TRUE;
ELSE
DisplayData[61].14:=FALSE;
END_IF
IF In2.15=FALSE THEN
DisplayData[61].15:=TRUE;
ELSE
DisplayData[61].15:=FALSE;
END_IF
IF In3.3=FALSE THEN
DisplayData[62].0:=TRUE;
ELSE
DisplayData[62].0:=FALSE;
END_IF
IF In3.4=FALSE THEN
DisplayData[62].1:=TRUE;
ELSE
DisplayData[62].1:=FALSE;
END_IF
IF In3.5=FALSE THEN
DisplayData[62].2:=TRUE;
ELSE
DisplayData[62].2:=FALSE;
END_IF
(*СВЯЗЬ В БВВ*)
IF Err[0]>0 THEN
DisplayData[60].1:=TRUE;
DisplayData[63].1:=FALSE;
ELSE
DisplayData[60].1:=FALSE;
DisplayData[63].1:=TRUE;
END_IF
IF Err[1]>0 THEN
DisplayData[60].2:=TRUE;
DisplayData[63].2:=FALSE;
ELSE
DisplayData[60].2:=FALSE;
DisplayData[63].2:=TRUE;
END_IF
IF Err[2]>0 THEN
DisplayData[60].3:=TRUE;
DisplayData[63].3:=FALSE;
ELSE
DisplayData[60].3:=FALSE;
DisplayData[63].3:=TRUE;
END_IF
IF Err[3]>0 THEN
DisplayData[60].4:=TRUE;
DisplayData[63].4:=FALSE;
ELSE
DisplayData[60].4:=FALSE;
DisplayData[63].4:=TRUE;
END_IF
IF Err[4]>0 THEN
DisplayData[60].5:=TRUE;
DisplayData[63].5:=FALSE;
ELSE
DisplayData[60].5:=FALSE;
DisplayData[63].5:=TRUE;
END_IF
(* НАРУШЕНИЕ СВЯЗИ АСШП *)
IF(In5.9 AND In5.10) OR (In5.9 AND In5.11) OR (In5.10 AND In5.11) OR (In5.9 AND In5.10 AND In5.11) THEN
DisplayData[60].6:=TRUE;
Out1:=0;
Out2.0:=FALSE;
Out2.1:=FALSE;
Out2.10:=FALSE;
Out2.11:=FALSE;
Out2.13:=FALSE;
DisplayData[63].6:=FALSE;
ELSE
DisplayData[60].6:=FALSE;
DisplayData[63].6:=TRUE;
END_IF 
END_FUNCTION

(* POU Link, ST *)
FUNCTION Link : BOOL
VAR_INPUT
END_VAR
VAR
	z: BYTE;
	a: BOOL;
	razrTON2: TON;
END_VAR
CASE NumberSend OF
0:
	     ModBusReadHoldReg[0](
		Enable:=TRUE ,
		Mode:=MB_RTU ,
		DevAddr:=1 ,
		FirstAddr:=1 ,
		Quantity:=1 ,
		ComHandle:=Settings.Port  ,
		TimeOut:=TimeOut,
		Buffer:=Buffer ,
		Complete=>Cmpl[0] ,
		Exception=>Err[0] ,
		ByteCnt=> );
	IF(cmpl[0]=TRUE) THEN
		IF (Err[0]=0) THEN
NumberSend:=1;
DisplayData[10].1:=TRUE;
			In1:=SHL(Buffer[0], 8)+Buffer[1];
		ELSE
NumberSend:=1;
DisplayData[10].1:=FALSE;
END_IF

END_IF
1:
 ModBusReadHoldReg[1](
		Enable:=TRUE ,
		Mode:=MB_RTU ,
		DevAddr:=2 ,
		FirstAddr:=1 ,
		Quantity:=1 ,
		ComHandle:=Settings.Port  ,
		TimeOut:=TimeOut,
		Buffer:=Buffer ,
		Complete=>Cmpl[1] ,
		Exception=>Err[1] ,
		ByteCnt=> );
	IF(cmpl[1]=TRUE) THEN
		IF (Err[1]=0) THEN
NumberSend:=2;
DisplayData[10].2:=TRUE;
			In2:=SHL(Buffer[0], 8)+Buffer[1];
		ELSE
NumberSend:=2;
DisplayData[10].2:=FALSE;
END_IF

END_IF
2:
 ModBusReadHoldReg[2](
		Enable:=TRUE ,
		Mode:=MB_RTU ,
		DevAddr:=3 ,
		FirstAddr:=1 ,
		Quantity:=1 ,
		ComHandle:=Settings.Port  ,
		TimeOut:=TimeOut,
		Buffer:=Buffer ,
		Complete=>Cmpl[2] ,
		Exception=>Err[2] ,
		ByteCnt=> );
	IF(cmpl[2]=TRUE) THEN
		IF (Err[2]=0) THEN
NumberSend:=3;
DisplayData[10].3:=TRUE;
			In3:=SHL(Buffer[0], 8)+Buffer[1];
		ELSE
NumberSend:=3;
DisplayData[10].3:=FALSE;
END_IF

END_IF
3:
 ModBusReadHoldReg[3](
		Enable:=TRUE ,
		Mode:=MB_RTU ,
		DevAddr:=4 ,
		FirstAddr:=1 ,
		Quantity:=1 ,
		ComHandle:=Settings.Port  ,
		TimeOut:=TimeOut,
		Buffer:=Buffer ,
		Complete=>Cmpl[3] ,
		Exception=>Err[3] ,
		ByteCnt=> );
	IF(cmpl[3]=TRUE) THEN
		IF (Err[3]=0) THEN
NumberSend:=4;
DisplayData[10].4:=TRUE;
			In4:=SHL(Buffer[0], 8)+Buffer[1];
		ELSE
NumberSend:=4;
DisplayData[10].4:=FALSE;
END_IF

END_IF
4:
 ModBusReadHoldReg[4](
		Enable:=TRUE ,
		Mode:=MB_RTU ,
		DevAddr:=5 ,
		FirstAddr:=1 ,
		Quantity:=1 ,
		ComHandle:=Settings.Port  ,
		TimeOut:=TimeOut,
		Buffer:=Buffer ,
		Complete=>Cmpl[4] ,
		Exception=>Err[4] ,
		ByteCnt=> );
	IF(cmpl[4]=TRUE) THEN
		IF (Err[4]=0) THEN
NumberSend:=5;
DisplayData[10].5:=TRUE;
			In5:=SHL(Buffer[0], 8)+Buffer[1];
		 ELSE
NumberSend:=5;
DisplayData[10].5:=FALSE;
END_IF

END_IF
5:
   Buffer[1]:=WORD_TO_BYTE(Out1 AND 16#00FF);
	       Buffer[0]:=WORD_TO_BYTE(SHR(Out1, 8));
	       ModBusWriteMultiReg[1](
		Enable:=TRUE ,
		Mode:=MB_RTU ,
		DevAddr:=1 ,
		FirstAddr:=0 ,
		Quantity:=1 ,
		ComHandle:=Settings.Port ,
		TimeOut:=TimeOut ,
		Buffer:=Buffer ,
			Complete=>Cmpl[5] ,
			Exception=>Err[5] ,
			RegCnt=> );
		IF(cmpl[5]=TRUE) THEN
		NumberSend:=6;
	END_IF
6:
  Buffer[1]:=WORD_TO_BYTE(Out2 AND 16#00FF);
	       Buffer[0]:=WORD_TO_BYTE(SHR(Out2, 8));
	       ModBusWriteMultiReg[2](
		Enable:=TRUE ,
		Mode:=MB_RTU ,
		DevAddr:=2 ,
		FirstAddr:=0 ,
		Quantity:=1 ,
		ComHandle:=Settings.Port ,
		TimeOut:=TimeOut ,
		Buffer:=Buffer ,
			Complete=>Cmpl[6] ,
			Exception=>Err[6] ,
			RegCnt=> );
		IF(cmpl[6]=TRUE) THEN
		NumberSend:=7;
	END_IF
7:
 Buffer[1]:=WORD_TO_BYTE(Out3 AND 16#00FF);
	       Buffer[0]:=WORD_TO_BYTE(SHR(Out3, 8));
	       ModBusWriteMultiReg[3](
		Enable:=TRUE ,
		Mode:=MB_RTU ,
		DevAddr:=3 ,
		FirstAddr:=0 ,
		Quantity:=1 ,
		ComHandle:=Settings.Port ,
		TimeOut:=TimeOut ,
		Buffer:=Buffer ,
			Complete=>Cmpl[7] ,
			Exception=>Err[7] ,
			RegCnt=> );
		IF(cmpl[7]=TRUE) THEN
		NumberSend:=8;
	END_IF
8:
 Buffer[1]:=WORD_TO_BYTE(Out4 AND 16#00FF);
	       Buffer[0]:=WORD_TO_BYTE(SHR(Out4, 8));
	       ModBusWriteMultiReg[3](
		Enable:=TRUE ,
		Mode:=MB_RTU ,
		DevAddr:=4 ,
		FirstAddr:=0 ,
		Quantity:=1 ,
		ComHandle:=Settings.Port ,
		TimeOut:=TimeOut ,
		Buffer:=Buffer ,
			Complete=>Cmpl[8] ,
			Exception=>Err[8] ,
			RegCnt=> );
		IF(cmpl[8]=TRUE) THEN
		NumberSend:=9;
	END_IF
9:
Buffer[1]:=WORD_TO_BYTE(Out5 AND 16#00FF);
	       Buffer[0]:=WORD_TO_BYTE(SHR(Out5, 8));
	       ModBusWriteMultiReg[3](
		Enable:=TRUE ,
		Mode:=MB_RTU ,
		DevAddr:=5 ,
		FirstAddr:=0 ,
		Quantity:=1 ,
		ComHandle:=Settings.Port ,
		TimeOut:=TimeOut ,
		Buffer:=Buffer ,
			Complete=>Cmpl[9] ,
			Exception=>Err[9] ,
			RegCnt=> );
		IF(cmpl[9]=TRUE) THEN
		NumberSend:=10;
	END_IF
10:
FOR z:=0 TO 90  BY 1 DO
		Buffer[z*2+1]:=WORD_TO_BYTE(DisplayData[z] AND 16#00FF);
		Buffer[z*2]:=WORD_TO_BYTE(SHR(DisplayData[z], 8));
	END_FOR
	ModBusWriteMultiReg[4](
		Enable:=TRUE ,
		Mode:=MB_RTU ,
		DevAddr:=10 ,
		FirstAddr:=300 ,
		Quantity:=65 ,
		ComHandle:=Settings.Port ,
		TimeOut:=T#100ms,
		Buffer:=Buffer ,
		Complete=>Cmpl[10] ,
		Exception=>Err[10] ,
		RegCnt=> );
	IF(cmpl[10]=TRUE) THEN
		NumberSend:=0;



	END_IF
END_CASE
END_FUNCTION
